{attribute 'GeneratedUsingTerminal: EK1122-0000-0018'}
{attribute addProperty BoxType "EK1122-0000-0018"}
{attribute addProperty Id "Beckhoff_EL68xxsub_EK1100EK1100_AB5A94672"}
{attribute addProperty CRC "1244082283"}
{attribute addProperty Size "2"}
TYPE Beckhoff_EL68xxEK1122_4A27306B EXTENDS EK1122_AB5A9467 :
STRUCT
	{attribute addProperty Name "Beckhoff_EL68xxsub_EK1100"}
	{attribute addProperty PreviousPort "Beckhoff EL68xxEK1122 : D"}
	Beckhoff_EL68xxsub_EK1100 : EK1100_AB5A9467;
END_STRUCT
END_TYPE

(* stored: Version 1.2.0.0, ProductVersion 3.1.4024.9
   DUT Beckhoff_EL68xxEK1122_4A27306B: Id {5080b004-3914-4364-80bc-65c7264552c3} *)
